TYPE M1AxialSupportProcesses :
STRUCT
	///Change a pressure setpoint, in Bar
	changePressureSetpoint: ChangeSetpointProcess;
	///Change the operating state of the pressure setpoint only
	changePressureSetpointState: ChangeOperatingStateProcess;
END_STRUCT
END_TYPE

(* stored: Version 1.1.0.1, ProductVersion 3.1.4019.2
   DUT M1AxialSupportProcesses: Id {b6c52f62-182d-4719-a5ad-0bf1ba501067} *)
